{attribute 'qualified_only'}
{attribute 'strict'}
TYPE PulsPisaChannelCount :
(
	Four := 4,
	Eight :=8
);
END_TYPE

(* stored: Version 1.1.0.1, ProductVersion 3.1.4024.15
   EnumerationTextList PulsPisaChannelCount: Id {48051dff-f5dc-4403-b486-271884baa014} *)
